{attribute 'qualified_only'}
{attribute 'global_init_slot' := '40500'}
VAR_GLOBAL
	Collection				: FB_ManagerCollection(0);
	Managers				: FB_ManagerAdapter(0);
END_VAR

(* stored: Version 1.1.0.1
   GVL GVL_Manager: Id {148d8567-00de-403f-8bdb-406acde852df} *)
